(* CoDeSys 2.3 export: CALC_FLAGS.EXP *)

(* POU lib/CALC_FLAGS, FBD *)
FUNCTION_BLOCK CALC_FLAGS
VAR_INPUT
	iSTATE								:	INT;
	xRESET							:	BOOL;
	xPART_START_POS				:	BOOL;
	xPUNCH_FULLY_EXTENDED	:	BOOL;
	xPART_END_POS				:	BOOL;
END_VAR
VAR_OUTPUT
	_xFLAG_PROCESSING_PART			:	BOOL;
	_xFLAG_ACCEPT_NEW_PART			:	BOOL;
	_xFLAG_ORIENTATION_CORRECT		:	BOOL;
END_VAR
VAR
	ft_partLeft						:	F_TRIG;
	rs_partOrientationCorrect		:	RS;
END_VAR
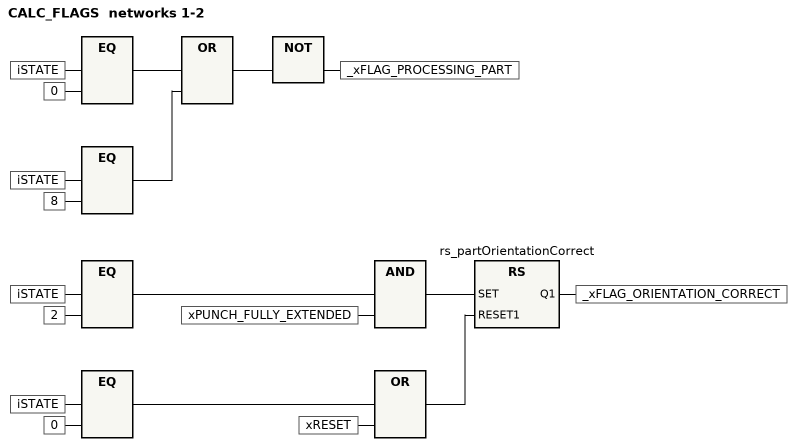
_FBD_ (* Function Block Diagram *)
NETWORK 1 processingPart: (* Determines if a part has entered or left and sets a flag accordingly. *)
	NOT(OR(EQ(iSTATE, 0), EQ(iSTATE, 8))) => _xFLAG_PROCESSING_PART
NETWORK 2 partOrientationCorrect: (* Checks if the Process at stage 2 determined that the part is in the correct orientation and sets the flag accordingly. *)
	rs_partOrientationCorrect:RS(SET: AND(EQ(iSTATE, 2), xPUNCH_FULLY_EXTENDED), RESET1: OR(EQ(iSTATE, 0), xRESET)) => _xFLAG_ORIENTATION_CORRECT
_END_FBD_
(* the same logic as Structured Text *)
(* Network 1: Determines if a part has entered or left and sets a flag accordingly. *)
processingPart:
_xFLAG_PROCESSING_PART := NOT ((iSTATE = 0) OR (iSTATE = 8));
(* Network 2: Checks if the Process at stage 2 determined that the part is in the correct orientation and sets the flag accordingly. *)
partOrientationCorrect:
rs_partOrientationCorrect(SET := (iSTATE = 2) AND xPUNCH_FULLY_EXTENDED, RESET1 := (iSTATE = 0) OR xRESET);
_xFLAG_ORIENTATION_CORRECT := rs_partOrientationCorrect.Q1;
END_FUNCTION_BLOCK
